{attribute 'linkalways'} 
{attribute 'no_explicit_call' := 'This FB is a CLASS and must be accessed using methods or properties'}
{attribute 'enable_dynamic_creation'}
FUNCTION_BLOCK ABSTRACT Node EXTENDS Disposable IMPLEMENTS I_Node
VAR
	_id : T_MAXSTRING;
	_order : DINT;
	_mode : DINT;
	eventEmitter : EventEmitter;
	inputPortHost : InputPortHost(eventEmitter);
	outputPortHost : OutputPortHost(eventEmitter);
	parameterHost : ParameterHost(eventEmitter);
	contentHost : ContentHost(eventEmitter);
	errorHost : ErrorHost(eventEmitter);
	extensionHost : ExtensionHost(eventEmitter);
	metadataHost : MetadataHost(eventEmitter);
END_VAR

METHOD PUBLIC Accept
VAR_INPUT
	Visitor : I_NodeVisitor;
END_VAR
Visitor.VisitNode(this^);
END_METHOD

METHOD AddContent
VAR_INPUT
	Content : I_Content;
END_VAR
contentHost.AddContent(Content);
END_METHOD

METHOD PUBLIC AddDataAsContent : I_Content;
VAR_INPUT
	Name : T_MAXSTRING;
	Data : I_Datatype;
END_VAR
AddDataAsContent := contentHost.AddDataAsContent(Name, Data);
END_METHOD

METHOD PUBLIC AddDataAsInputPort : I_InputPort;
VAR_INPUT
	Name : T_MAXSTRING;
	Data : I_Datatype;
END_VAR
AddDataAsInputPort := inputPortHost.AddDataAsInputPort(Name, Data);
END_METHOD

METHOD PUBLIC AddDataAsMetadata : I_Metadata;
VAR_INPUT
	Name : T_MAXSTRING;
	Data : I_Datatype;
END_VAR
AddDataAsMetadata := metadataHost.AddDataAsMetadata(Name, Data);
END_METHOD

METHOD PUBLIC AddDataAsOutputPort : I_OutputPort;
VAR_INPUT
	Name : T_MAXSTRING;
	Data : I_Datatype;
END_VAR
AddDataAsOutputPort := outputPortHost.AddDataAsOutputPort(Name, Data);
END_METHOD

METHOD PUBLIC AddDataAsParameter : I_Parameter;
VAR_INPUT
	Name : T_MAXSTRING;
	Data : I_Datatype;
END_VAR
AddDataAsParameter := parameterHost.AddDataAsParameter(Name, Data);
END_METHOD

METHOD AddError
VAR_INPUT
	Error : I_Error;
END_VAR
errorHost.AddError(Error);
END_METHOD

METHOD AddExtension
VAR_INPUT
	Extension : I_Extension;
END_VAR
extensionHost.AddExtension(Extension);
END_METHOD

METHOD AddInputPort
VAR_INPUT
	InputPort : I_InputPort;
END_VAR
inputPortHost.AddInputPort(InputPort);
END_METHOD

METHOD AddMetadata
VAR_INPUT
	Metadata : I_Metadata;
END_VAR
metadataHost.AddMetadata(Metadata);
END_METHOD

METHOD AddOutputPort
VAR_INPUT
	OutputPort : I_OutputPort;
END_VAR
outputPortHost.AddOutputPort(OutputPort);
END_METHOD

METHOD AddParameter
VAR_INPUT
	Parameter : I_Parameter;
END_VAR
parameterHost.AddParameter(Parameter);
END_METHOD

METHOD PUBLIC ABSTRACT Clone : I_Node
VAR_INPUT
END_VAR
END_METHOD

METHOD PROTECTED EmitNodeExecuteBeginEvent : BOOL;
VAR
	pNodeExecuteBeginEvent : POINTER TO NodeExecuteBeginEvent;
END_VAR
pNodeExecuteBeginEvent := __NEW(NodeExecuteBeginEvent(TargetNode := THIS^));
eventEmitter.Emit('OnNodeExecuteBegin',pNodeExecuteBeginEvent^);
pNodeExecuteBeginEvent^.Dispose();
END_METHOD

METHOD PROTECTED EmitNodeExecuteEndEvent : BOOL;
VAR
	pNodeExecuteEndEvent : POINTER TO NodeExecuteEndEvent;
END_VAR
pNodeExecuteEndEvent := __NEW(NodeExecuteEndEvent(TargetNode := THIS^));
eventEmitter.Emit('OnNodeExecuteEnd',pNodeExecuteEndEvent^);
pNodeExecuteEndEvent^.Dispose();
END_METHOD

METHOD PROTECTED EmitOnNodePreExecuteEvent : BOOL;
VAR_INPUT
	CancelRequested : REFERENCE TO BOOL;
END_VAR
VAR
	pNodePreExecuteEvent : POINTER TO NodePreExecuteEvent;
END_VAR
pNodePreExecuteEvent := __NEW(NodePreExecuteEvent(TargetNode := THIS^));
eventEmitter.Emit('OnNodePreExecute',pNodePreExecuteEvent^);

IF pNodePreExecuteEvent^.ExecuteCancelled THEN
	CancelRequested := TRUE;
END_IF

pNodePreExecuteEvent^.Dispose();
END_METHOD

METHOD PUBLIC Execute
VAR
	cancelExecuteResponse : BOOL := FALSE;
END_VAR
EmitOnNodePreExecuteEvent(cancelExecuteResponse);

IF cancelExecuteResponse THEN
	RETURN;
END_IF

EmitNodeExecuteBeginEvent();
OnExecute();
EmitNodeExecuteEndEvent();
END_METHOD

METHOD FB_init : BOOL
VAR_INPUT
	bInitRetains : BOOL; // if TRUE, the retain variables are initialized (warm start / cold start)
	bInCopyCode : BOOL;  // if TRUE, the instance afterwards gets moved into the copy code (online change)
END_VAR
InitializeNode(this^);
END_METHOD

PROPERTY PUBLIC Id : T_MAXSTRING
GET
Id := _id;
END_GET
END_PROPERTY

METHOD PROTECTED InitializeNode
VAR_INPUT
	Self : I_Node;
END_VAR
END_METHOD

PROPERTY PUBLIC Mode : DINT
GET
Mode := _mode;
END_GET
END_PROPERTY

METHOD PUBLIC OffEvent
VAR_INPUT
	EventName : T_MaxString;
	EventHandler : I_EventHandler;
END_VAR
eventEmitter.OffEvent(EventName, EventHandler);
END_METHOD

METHOD PUBLIC OnceEvent
VAR_INPUT
	EventName : T_MaxString;
	EventHandler : I_EventHandler;
END_VAR
eventEmitter.OnceEvent(EventName, EventHandler);
END_METHOD

METHOD PUBLIC OnEvent
VAR_INPUT
	EventName : T_MaxString;
	EventHandler : I_EventHandler;
END_VAR
eventEmitter.OnEvent(EventName, EventHandler);
END_METHOD

METHOD PROTECTED ABSTRACT OnExecute : HRESULT
END_METHOD

PROPERTY PUBLIC Order : DINT
GET
Order := _order;
END_GET
END_PROPERTY

METHOD PUBLIC SerializeWith
VAR_INPUT
	Serializer : I_Serializer;
END_VAR
Serializer.StartObject();
inputPortHost.SerializeWith(Serializer);
outputPortHost.SerializeWith(Serializer);
parameterHost.SerializeWith(Serializer);
contentHost.SerializeWith(Serializer);
errorHost.SerializeWith(Serializer);
extensionHost.SerializeWith(Serializer);
metadataHost.SerializeWith(Serializer);
Serializer.EndObject();
END_METHOD

METHOD PUBLIC TryDeserializeFrom : BOOL
VAR_INPUT
	Deserializer : I_Deserializer;
END_VAR
TryDeserializeFrom := 
	Deserializer.TryGetKeyString('id', _id) AND
	Deserializer.TryGetKeyDint('order', _order) AND
	Deserializer.TryGetKeyDint('mode', _mode) AND
	parameterHost.TryDeserializeFrom(Deserializer) AND 
	extensionHost.TryDeserializeFrom(Deserializer);
END_METHOD

METHOD PUBLIC TryGetContentByName : BOOL
VAR_INPUT
	Name : T_MAXSTRING;
	Destination : REFERENCE TO I_Content;
END_VAR
VAR
	extensionName : T_MAXSTRING;
	extension : I_Extension;
	contentName : T_MAXSTRING;
END_VAR
IF Not HasExtensionNamespace(Name) THEN
	TryGetContentByName := contentHost.TryGetContentByName(Name,Destination);
	RETURN;
END_IF

extensionName := RemoveLastSegmentFromNamespace(Name);
contentName := GetLastSegmentFromNamespace(Name);

IF NOT TryGetExtensionByName(extensionName, extension) THEN
	RETURN;
END_IF

TryGetContentByName := extension.TryGetContentByName(contentName, Destination);
END_METHOD

METHOD PUBLIC TryGetExtensionByName : BOOL
VAR_INPUT
	Name : T_MAXSTRING;
	Destination : REFERENCE TO I_Extension;
END_VAR
TryGetExtensionByName := extensionHost.TryGetExtensionByName(Name, Destination);
END_METHOD

METHOD PUBLIC TryGetInputPortByName : BOOL
VAR_INPUT
	Name : T_MAXSTRING;
	Destination : REFERENCE TO I_InputPort;
END_VAR
VAR
	extensionName : T_MAXSTRING;
	extension : I_Extension;
	portName : T_MAXSTRING;
END_VAR
IF NOT HasExtensionNamespace(Name) THEN
	TryGetInputPortByName := inputPortHost.TryGetInputPortByName(Name,Destination);
	RETURN;
END_IF

extensionName := RemoveLastSegmentFromNamespace(Name);
portName := GetLastSegmentFromNamespace(Name);

IF NOT TryGetExtensionByName(extensionName, extension) THEN
	RETURN;
END_IF

TryGetInputPortByName := extension.TryGetInputPortByName(portName, Destination);
END_METHOD

METHOD PUBLIC TryGetMetadataByName : BOOL
VAR_INPUT
	Name : T_MAXSTRING;
	Destination : REFERENCE TO I_Metadata;
END_VAR
VAR
	extensionName : T_MAXSTRING;
	extension : I_Extension;
	metadatumName : T_MAXSTRING;
END_VAR
IF NOT HasExtensionNamespace(Name) THEN
	TryGetMetadataByName := metadataHost.TryGetMetadataByName(Name,Destination);
	RETURN;
END_IF

extensionName := RemoveLastSegmentFromNamespace(Name);
metadatumName := GetLastSegmentFromNamespace(Name);

IF NOT TryGetExtensionByName(extensionName, extension) THEN
	RETURN;
END_IF

TryGetMetadataByName := extension.TryGetMetadataByName(metadatumName, Destination);
END_METHOD

METHOD PUBLIC TryGetOutputPortByName : BOOL
VAR_INPUT
	Name : T_MAXSTRING;
	Destination : REFERENCE TO I_OutputPort;
END_VAR
VAR
	extensionName : T_MAXSTRING;
	extension : I_Extension;
	portName : T_MAXSTRING;
END_VAR
IF NOT HasExtensionNamespace(Name) THEN
	TryGetOutputPortByName := outputPortHost.TryGetOutputPortByName(Name,Destination);
	RETURN;
END_IF

extensionName := RemoveLastSegmentFromNamespace(Name);
portName := GetLastSegmentFromNamespace(Name);

IF NOT TryGetExtensionByName(extensionName, extension) THEN
	RETURN;
END_IF

TryGetOutputPortByName := extension.TryGetOutputPortByName(portName, Destination);
END_METHOD

METHOD PUBLIC TryGetParameterByName : BOOL
VAR_INPUT
	Name : T_MAXSTRING;
	Destination : REFERENCE TO I_Parameter;
END_VAR
VAR
	extensionName : T_MAXSTRING;
	extension : I_Extension;
	parameterName : T_MAXSTRING;
END_VAR
IF Not HasExtensionNamespace(Name) THEN
	TryGetParameterByName := parameterHost.TryGetParameterByName(Name,Destination);
	RETURN;
END_IF

extensionName := RemoveLastSegmentFromNamespace(Name);
parameterName := GetLastSegmentFromNamespace(Name);

IF NOT TryGetExtensionByName(extensionName, extension) THEN
	RETURN;
END_IF

TryGetParameterByName := extension.TryGetParameterByName(parameterName, Destination);
END_METHOD

END_FUNCTION_BLOCK

(* stored: Version 1.1.0.1, ProductVersion 3.1.4024.12
   POU Node: Id {8b8910db-ad72-05a5-0556-4fd11e61a0b6}, SpecialFunc None
   Folder Abstract: Id {dbd4d2fd-33d8-0c09-0e75-48a8aa9fa6b2}
   Folder Constructor: Id {a1653d54-8e94-41a9-8c14-cce7fd0b4618}
   Folder Protected: Id {f0af3386-ca84-0b52-03e7-a20a015d9afb}
   Method Accept: Id {4230f410-f451-039d-2604-d2edaf4d13f7}
   Method AddContent: Id {c0b648e0-1253-452b-90ed-e8143a2d89de}
   Method AddDataAsContent: Id {892184f4-5f52-4626-821f-5a3491889bf3}
   Method AddDataAsInputPort: Id {bf7b53bb-ee8c-454b-9fed-7549fb092389}
   Method AddDataAsMetadata: Id {27de0cd1-b5b3-4c95-81d1-bae2f0aa4ba2}
   Method AddDataAsOutputPort: Id {67754854-46b8-493e-aa68-90f8cff784b2}
   Method AddDataAsParameter: Id {369f41f2-8c43-4545-92b8-386c840b633c}
   Method AddError: Id {68a33ee7-a8d2-4500-8be9-00fe1a233658}
   Method AddExtension: Id {3c2efc0a-31a2-4144-a0f8-6a9d285ba29e}
   Method AddInputPort: Id {f3d8ee87-5b7a-4f8c-afb8-98ced33fe48d}
   Method AddMetadata: Id {0f29f336-eda4-437c-a7a8-83e334c02d43}
   Method AddOutputPort: Id {baff6e52-981c-417b-a16e-c84e80784dd2}
   Method AddParameter: Id {697d49dc-f6b8-4cfb-981a-457bda0c8dd7}
   Method Clone: Id {026c4113-8518-4d67-89a7-84bf1813f983}
   Method EmitNodeExecuteBeginEvent: Id {446e8833-be75-08b5-20ae-de0735b20b11}
   Method EmitNodeExecuteEndEvent: Id {a7ad8910-3e19-0f65-0e88-7dce16ea71b6}
   Method EmitOnNodePreExecuteEvent: Id {78e8301b-1d71-0189-3c20-c1b779dc4500}
   Method Execute: Id {d408825d-3e00-0ecb-23c4-0596c3d88698}
   Method FB_init: Id {f4087af8-03a6-4168-ab7f-e8de08c6cd17}
   Property Id: Id {83736b4e-b1bc-0adb-2e43-a65e1cb4d5a3}
   Get Get: Id {e5d6cfcc-06b4-0c3a-347e-7067097be358}
   Method InitializeNode: Id {01545b32-13d6-40b0-b942-2e82aaf63024}
   Property Mode: Id {7c0c904d-4b3b-026a-34c8-a61976b560fb}
   Get Get: Id {e082d771-5c44-02f0-0e53-87177d47eeff}
   Method OffEvent: Id {31f72dc9-3d1e-4ce4-bd2f-cdb6bf6d0c73}
   Method OnceEvent: Id {4033b450-0033-49f9-8e3c-0af1c515fb9e}
   Method OnEvent: Id {f228b5cc-83e5-4635-9fa1-3741721a5186}
   Method OnExecute: Id {3305d23e-f58f-0290-011d-0ef3d43fdad1}
   Property Order: Id {b8b6cab5-3d18-0865-3a46-18681789df72}
   Get Get: Id {0242dc0d-dd4a-0656-266d-688e1d427b8a}
   Method SerializeWith: Id {34e53c74-e83e-4449-a443-ad491ecc1661}
   Method TryDeserializeFrom: Id {b10f689b-9a8b-4119-b4c9-ae83d038092d}
   Method TryGetContentByName: Id {a442af03-1b8f-4c53-817a-0af473a480df}
   Method TryGetExtensionByName: Id {f31010b5-cd16-4ab4-8e30-e0b827c31eb1}
   Method TryGetInputPortByName: Id {97da5ea4-1784-4901-aa96-8e03ff2613bf}
   Method TryGetMetadataByName: Id {37dc25b0-8e02-4776-a290-bac7c8fa7609}
   Method TryGetOutputPortByName: Id {5e09a92c-9cf0-4b12-abd1-c4e11e5fff8d}
   Method TryGetParameterByName: Id {168c4d2c-f9f8-420d-bb40-e4bd5929ea86} *)
